% RSLogix 500 project MUX.RSS, saved by version 8.30.00.16 %
PROJECT "UNTITLED"    % processor: Bul.1763 MicroLogix 1100 Series B %

PROGRAM FILES
  LAD 2   2 rungs

DATA FILES
  O0 OUTPUT  4 elements
  I1 INPUT  6 elements
  S2 STATUS  66 elements
  B3 BINARY  1 elements
  T4 TIMER  1 elements
  C5 COUNTER  1 elements
  R6 CONTROL  1 elements
  N7 INTEGER  1 elements
  F8 FLOAT  1 elements

LADDER 2
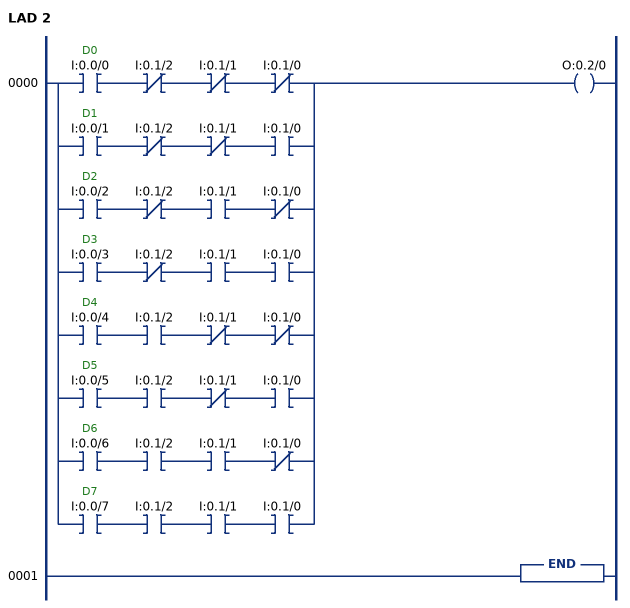
% Rung: 0 %
SOR BST XIC I:0.0/0 XIO I:0.1/2 XIO I:0.1/1 XIO I:0.1/0 NXB XIC I:0.0/1 XIO I:0.1/2 XIO I:0.1/1 XIC I:0.1/0 NXB XIC I:0.0/2 XIO I:0.1/2 XIC I:0.1/1 XIO I:0.1/0 NXB XIC I:0.0/3 XIO I:0.1/2 XIC I:0.1/1 XIC I:0.1/0 NXB XIC I:0.0/4 XIC I:0.1/2 XIO I:0.1/1 XIO I:0.1/0 NXB XIC I:0.0/5 XIC I:0.1/2 XIO I:0.1/1 XIC I:0.1/0 NXB XIC I:0.0/6 XIC I:0.1/2 XIC I:0.1/1 XIO I:0.1/0 NXB XIC I:0.0/7 XIC I:0.1/2 XIC I:0.1/1 XIC I:0.1/0 BND OTE O:0.2/0 EOR
%   I:0.0/0  D0 %
%   I:0.0/1  D1 %
%   I:0.0/2  D2 %
%   I:0.0/3  D3 %
%   I:0.0/4  D4 %
%   I:0.0/5  D5 %
%   I:0.0/6  D6 %
%   I:0.0/7  D7 %
% Rung: 1 %
SOR END EOR
